{attribute 'enable_dynamic_creation' := ''}
FUNCTION_BLOCK Realsubject IMPLEMENTS Subject_Interface
VAR
	///Variable to get and set values
	iProp: INT;
END_VAR

METHOD Get_Method : INT
//Asks for the value of the object's iProp variable and passes it to the caller

Get_Method := THIS^.iProp;
END_METHOD

METHOD Set_Method
VAR_INPUT
	///Value to be set on the iProp varible of realSubjectInstance
	num: INT;
END_VAR
//Stores the value of the caller object on iProp variable. 

THIS^.iProp := num;
END_METHOD

END_FUNCTION_BLOCK

(* stored: Version 1.1.0.1, ProductVersion 3.1.4024.12
   POU Realsubject: Id {b98cd672-9806-4c71-939e-f49997b14c1b}, SpecialFunc None
   Method Get_Method: Id {e5d61f1d-ce40-49a3-b00d-81878706227a}
   Method Set_Method: Id {d1c85d57-484f-4462-b13a-610d0968786b} *)
